FUNCTION_BLOCK AUDI_CTUD_UDINT (* Event-Driven Up-Down Counter *)
  (* Standard: 61499-1-A.x; Classification: Event-driven blocks; Function: Up-Down-counter; Description: Copyright (c) 2017, 2024 fortiss GmbH, JKU, HR Agrartechnik GmbH This program and the accompanying materials are made available under the terms of the Eclipse Public License 2.0 which is available at https://www.eclipse.org/legal/epl-2.0/ SPDX-License-Identifier: EPL-2.0 *)
  (* Version 3.0, 2025-04-14, Franz Höpfinger, HR Agrartechnik GmbH, Made Version 3.0.0 inspired by Work from Patrick Aigner *)
  (* Version 1.2, 2024-02-10, Franz Höpfinger, HR Agrartechnik GmbH, Copy over E_CTUD to E_CTUD_UDINT *)
  (* Version 1.1, 2019-07-09, Alois Zoitl, JKU, fixed bug in down counting (E_CTUD) *)
  (* Version 1.0, 2017-09-22, Alois Zoitl, fortiss GmbH, initial API and implementation and/or initial documentation (E_CTUD) *)
  PACKAGE iec61499::events;
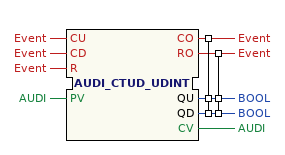
  EVENT_INPUT
    CU; (* Count Up *)
    CD; (* Count Down *)
    R; (* Reset *)
  END_EVENT
  EVENT_OUTPUT
    CO WITH QU, QD; (* Count Output Event *)
    RO WITH QU, QD; (* Reset Output Event *)
  END_EVENT
  VAR_OUTPUT
    QU : BOOL; (* CV >=PV *)
    QD : BOOL; (* CV <= 0 *)
  END_VAR
  SOCKETS
    PV : adapter::types::unidirectional::AUDI; (* Preset Value *)
  END_SOCKETS
  PLUGS
    CV : adapter::types::unidirectional::AUDI; (* Counter Value *)
  END_PLUGS
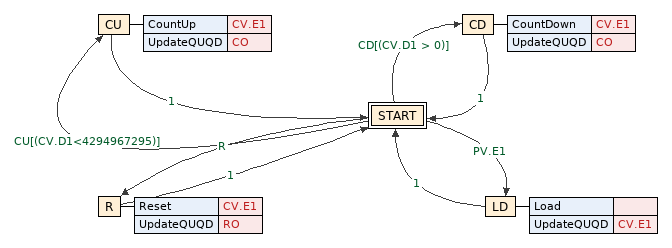
  EC_STATES
    START;
    CU : CountUp -> CV.E1, UpdateQUQD -> CO;
    R : Reset -> CV.E1, UpdateQUQD -> RO;
    CD : CountDown -> CV.E1, UpdateQUQD -> CO;
    LD : Load, UpdateQUQD -> CV.E1;
  END_STATES
  EC_TRANSITIONS
    START TO CU := CU[(CV.D1<4294967295)];
    CU TO START := 1;
    START TO R := R;
    R TO START := 1;
    START TO CD := CD[(CV.D1 > 0)];
    CD TO START := 1;
    START TO LD := PV.E1;
    LD TO START := 1;
  END_TRANSITIONS
  ALGORITHM CountUp IN ST:
CV.D1 := CV.D1 + 1;
  END_ALGORITHM
  ALGORITHM Reset IN ST:
CV.D1 := 0;
  END_ALGORITHM
  ALGORITHM Load IN ST:
CV.D1 := PV.D1;
  END_ALGORITHM
  ALGORITHM UpdateQUQD IN ST:
QU := (CV.D1 >= PV.D1);
QD := (CV.D1 = 0);
  END_ALGORITHM
  ALGORITHM CountDown IN ST:
CV.D1 := CV.D1 - 1;
  END_ALGORITHM
END_FUNCTION_BLOCK
